FUNCTION F_BuildHttpPostRequest : UDINT
VAR_INPUT
	i_pHttpRequest 		: POINTER TO ST_HTTP_Request;
	i_stHttpConnParams	: ST_HTTP_Connection_Parameters;
END_VAR
VAR_IN_OUT
	io_arrBytesToSend	: ARRAY[0..HTTP_SEND_DATA_ARRAY_SIZE] OF BYTE;
END_VAR
VAR
	sData				: T_MaxString;
	i					: INT;
	nContentLength		: DINT;
	fbBinaryWriter		: FB_BinaryWriter;
	sRequestString		: STRING(255);
END_VAR


fbBinaryWriter.Init(ADR(io_arrBytesToSend), SIZEOF(io_arrBytesToSend));
MEMSET(ADR(io_arrBytesToSend), 0, SIZEOF(io_arrBytesToSend));

fbBinaryWriter.WriteString('POST ');
fbBinaryWriter.WriteString(i_stHttpConnParams.sRequestURI);
fbBinaryWriter.WriteString(' HTTP/1.0$R$N'); // Lets use HTTP 1.0 because responce with "Transfer-Encoding:chunked is much more complex to parse
fbBinaryWriter.WriteString('Host: ');
fbBinaryWriter.WriteString(i_stHttpConnParams.sHostName);
fbBinaryWriter.WriteString(' $R$N');
fbBinaryWriter.WriteString('User-Agent: TwinCAT HttpClient$R$N');
fbBinaryWriter.WriteString('Content-Type: application/x-www-form-urlencoded$R$N');

// Calculate the length of data
FOR i := 0 TO UDINT_TO_INT(HTTP_PARAMETERS_ARRAY_SIZE) DO 
	IF LEN(i_pHttpRequest^.arrParameters[i].sName) > 0 THEN
		IF i > 0 THEN nContentLength := nContentLength + 1; END_IF
		nContentLength := nContentLength + LEN(i_pHttpRequest^.arrParameters[i].sName) + LEN(i_pHttpRequest^.arrParameters[i].sValue) + 1;
	END_IF
END_FOR	

fbBinaryWriter.WriteString(CONCAT('Content-Length: ', DINT_TO_STRING(nContentLength)));


// Http request headers always end to double new line		
fbBinaryWriter.WriteString('$R$N$R$N');

// Write the POST data into request body
FOR i := 0 TO UDINT_TO_INT(HTTP_PARAMETERS_ARRAY_SIZE) DO 
	IF LEN(i_pHttpRequest^.arrParameters[i].sName) > 0 THEN
		IF i > 0 THEN fbBinaryWriter.WriteString('&'); END_IF
		fbBinaryWriter.WriteString(i_pHttpRequest^.arrParameters[i].sName);
		fbBinaryWriter.WriteString('=');
		fbBinaryWriter.WriteString(i_pHttpRequest^.arrParameters[i].sValue);
	END_IF
END_FOR

// Http request body always ends to new line		
fbBinaryWriter.WriteString('$R$N');


sRequestString := fbBinaryWriter.ToString;
F_BuildHttpPostRequest := fbBinaryWriter.Length;

(****** POST Request principle ***********************************************************************

sPostData = 'param1=1&param2=2&param3=3';
fbBinaryWriter.WriteString('POST /demot/rest-demo/ HTTP/1.1$R$N');
fbBinaryWriter.WriteString('Host: bafdemo.cloudapp.net $R$N');
fbBinaryWriter.WriteString('User-Agent: TwinCAT 3.1$R$N');
fbBinaryWriter.WriteString('Content-Type: application/x-www-form-urlencoded$R$N');
fbBinaryWriter.WriteString(CONCAT('Content-Length: ', DINT_TO_STRING(LEN(sPostData))));
fbBinaryWriter.WriteString('$R$N$R$N');
fbBinaryWriter.WriteString(sPostData);
fbBinaryWriter.WriteString('$R$N');

******************************************************************************************************)

END_FUNCTION

(* stored: Version 1.1.0.1, ProductVersion 3.1.4020.12
   POU F_BuildHttpPostRequest: Id {e0e8ac94-2d97-4d93-b824-054fc419956a}, SpecialFunc None *)
